PROGRAM pouAxis
VAR
END_VAR

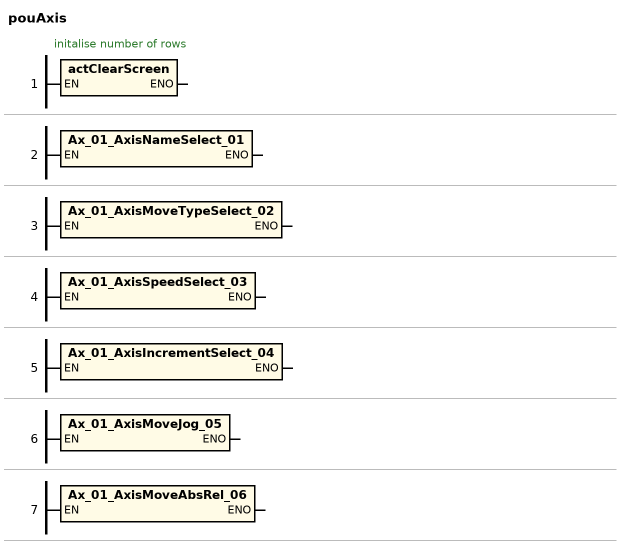
// NETWORK 1
// initalise number of rows
actClearScreen();

// NETWORK 2
Ax_01_AxisNameSelect_01();

// NETWORK 3
Ax_01_AxisMoveTypeSelect_02();

// NETWORK 4
Ax_01_AxisSpeedSelect_03();

// NETWORK 5
Ax_01_AxisIncrementSelect_04();

// NETWORK 6
Ax_01_AxisMoveJog_05();

// NETWORK 7
Ax_01_AxisMoveAbsRel_06();

ACTION actClearScreen:
//clear HMI row for manual insertion
HMIData.gAxisRows.gMotionRow1.IndexLocation := 0;
HMIData.gAxisRows.gMotionRow2.IndexLocation := 20;
HMIData.gAxisRows.gMotionRow3.IndexLocation := 40;
HMIData.gAxisRows.gMotionRow4.IndexLocation := 60;
HMIData.gAxisRows.gMotionRow5.IndexLocation := 80;
HMIData.gAxisRows.gMotionRow6.IndexLocation := 100;

//clear axis row layout
HMIData.gAxisNumRows := 0;
END_ACTION

END_PROGRAM

(* stored: Version 1.1.0.1, ProductVersion 3.1.4024.12
   POU pouAxis: Id {0a1eb7e7-2ca7-4349-8d96-78253461d98b}, SpecialFunc None
   Action actClearScreen: Id {a9ff748a-de6a-4eb1-8d41-a39e8e6638f7} *)
